INTERFACE I_TriggerPort

PROPERTY PUBLIC Result : HRESULT
GET
END_GET
END_PROPERTY

END_INTERFACE

(* stored: Version 1.1.0.1, ProductVersion 3.1.4024.12
   Itf I_TriggerPort: Id {bb9f66be-c1da-0d9a-2dcd-8055d5a33ccd}
   Property Result: Id {286a36f1-5b95-0eff-056d-234ef6fafb58}
   Get Get: Id {737437ec-47f7-005b-2502-26bc66e9b00d} *)
